(* IEC 61131-3 sources: structured-text/samples/unsupported/invalid_decl_type, 7 files *)

(* ---- f.11.st ---- *)
FUNCTION ALRMINT : BOOL
VAR_INPUT
  IN:INT;
  THI:INT ;
  TLO:INT  ;
END_VAR
VAR_OUTPUT
  HI: BOOL;
  LO: BOOL;
END_VAR
HI := IN > THI ;

LO := IN < THL ;
ALRMINT := THI OR THL ;
END_FUNCTION

(* ---- f10.st ---- *)
FUNCTION SIMPLE_FUN : REAL
    VAR_INPUT
  		A, B : REAL ;
      	C : REAL := 1.0;
  	END_VAR
  	VAR_IN_OUT COUNT : INT ; END_VAR
  	VAR COUNTP1 : INT ; END_VAR

  	COUNTP1 := ADD(COUNT,1);
  	COUNT := COUNTP1 ;
    SIMPLE_FUN := A*B/C;
END_FUNCTION

(* ---- f5.st ---- *)
FUNCTION Test : INT
	VAR_INPUT
		B, C, D : INT;
		X : INT;
	END_VAR
	VAR_OUTPUT
		A : INT;
		NO_ERR : BOOL;
	END_VAR

	A := ADD(B, C, D);
	A := SHL(IN:=B, N:=C);
	A := SHL(EN:=ENABLE, IN:=B, N:=C, NOT ENO=>NO_ERR);
	A := INC(V:=X);

END_FUNCTION

(* ---- t19-1.st ---- *)
FUNCTION Test : INT
	VAR_INPUT
		B, COND, TEMPL : INT;
	END_VAR
	VAR_OUTPUT
		A : INT;
	END_VAR

	A := LIMIT(EN:=COND, IN:=B, MX:=5, ENO=>TEMPL);

END_FUNCTION

(* ---- t19-2.st ---- *)
FUNCTION Test : INT
	VAR_INPUT
		B : INT;
	END_VAR
	VAR_OUTPUT
		A : INT;
	END_VAR

	A := LIMIT(1, B, 5);

END_FUNCTION

(* ---- t56-1.st ---- *)
FUNCTION Test : INT
	VAR_INPUT
		B : INT;
	END_VAR
	VAR_OUTPUT
		A, CV : INT;
		C : REAL;
	END_VAR

	A := B;
	CV := CV+1;
	C := SIN(X);

END_FUNCTION

(* ---- t56-4.st ---- *)
FUNCTION Test : BOOL
	VAR_INPUT
		A, B, C : REAL;
	END_VAR
	VAR_OUTPUT
		D, X1, X2 : REAL;
		NROOTS : INT;
	END_VAR

	D := B*B - 4*A*C ;
	IF D < 0.0 THEN NROOTS := 0 ;
	ELSIF D = 0.0 THEN
		NROOTS := 1 ;
		X1 := - B/(2.0*A) ;
	ELSE
		NROOTS := 2 ;
		X1 := (- B + SQRT(D))/(2.0*A) ;
		X2 := (- B - SQRT(D))/(2.0*A) ;
	END_IF ;
END_FUNCTION
